{attribute 'qualified_only'}
VAR_GLOBAL
	Plant_B57_Control : PlantAndCMs.Udt_PlantControl;
	
	Plant_B28_Control : PlantAndCMs.Udt_PlantControl;
END_VAR

(* stored: Version 1.1.0.1, ProductVersion 3.1.4024.13
   GVL CMD: Id {70f5f6d9-35db-4032-a601-50bccae1941c} *)
